// TIA Portal project "Project34" (V11)

(* hardware
DEVICE "S7-400 station_1"  S7400.Device
   slot 0: "UR1_0"  UR1  6ES7 400-1TA01-0AA0
   slot 2: "PLC_1"  Unspecific CPU S7 400  6ES7 4XX XXXXX XXXX
*)

// ===== PLC "PLC_1"  Unspecific CPU S7 400 =====

VAR_GLOBAL   // PLC tag table "Default tag table"
   "s1" AT %I0.0 : Bool;
   "s2" AT %I0.1 : Bool;
   "k2" AT %Q0.3 : Bool;
   "b2" AT %I0.3 : Bool;
   "k1" AT %Q0.2 : Bool;
   "Tag_1" AT %T1 : Timer;
   "b1" AT %I0.2 : Bool;
   "Tag_3" AT %T2 : Timer;
   "h1" AT %Q0.0 : Bool;
   "h2" AT %Q0.1 : Bool;
END_VAR

ORGANIZATION_BLOCK "Main"   // OB1, LAD
TITLE = "Main Program Sweep (Cycle)"
{ S7_Optimized_Access := 'FALSE' }
VERSION : 0.1
   VAR_TEMP
      OB1_EV_CLASS : Byte;   // Bits 0-3 = 1 (Coming event), Bits 4-7 = 1 (Event class 1)
      OB1_SCAN_1 : Byte;   // 1 (Cold restart scan 1 of OB 1), 3 (Scan 2-n of OB 1)
      OB1_PRIORITY : Byte;   // Priority of OB Execution
      OB1_OB_NUMBR : Byte;   // 1 (Organization block 1, OB1)
      OB1_RESERVED_1 : Byte;   // Reserved for system
      OB1_RESERVED_2 : Byte;   // Reserved for system
      OB1_PREV_CYCLE : Int;   // Cycle time of previous OB1 scan (milliseconds)
      OB1_MIN_CYCLE : Int;   // Minimum cycle time of OB1 (milliseconds)
      OB1_MAX_CYCLE : Int;   // Maximum cycle time of OB1 (milliseconds)
      OB1_DATE_TIME : Date_And_Time;   // Date and time OB1 started
   END_VAR
   VAR_TEMP   // added for the SCL form of the ladder/FBD networks
      _w1 : Bool;
      _s5time1 : S5Time;
   END_VAR
BEGIN

REGION Network 1
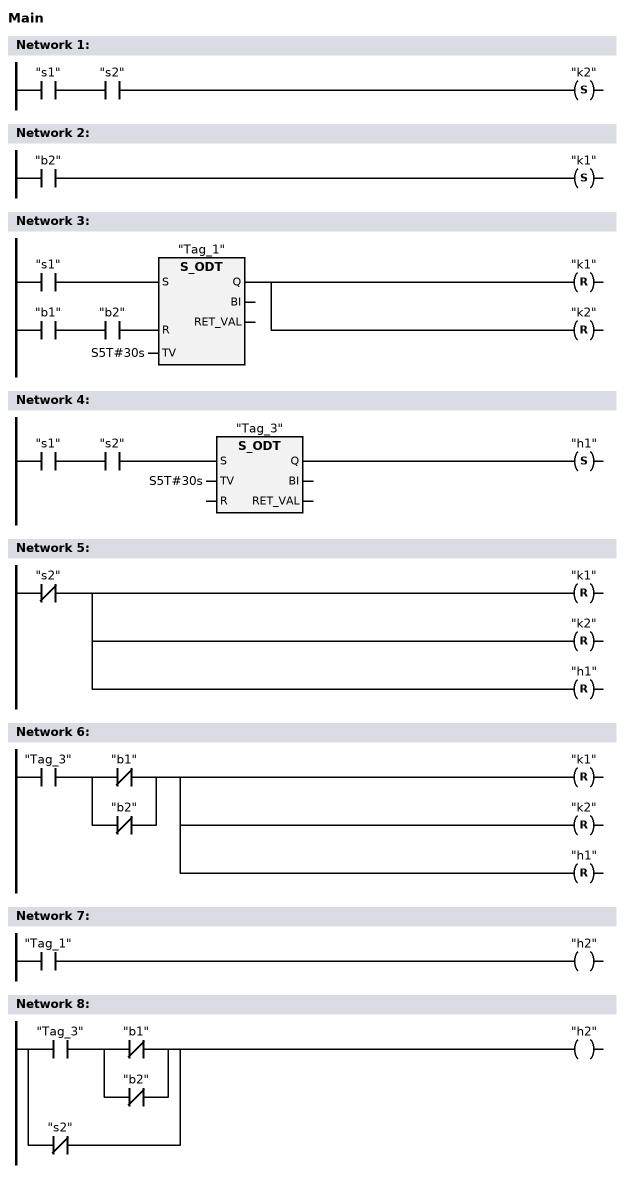
   RUNG wire#powerrail
      Contact( "s1" )
      Contact( "s2" )
      S_Coil( "k2" )
   END_RUNG
   // the same network as SCL:
   IF "s1" AND "s2" THEN "k2" := TRUE; END_IF;
END_REGION

REGION Network 2
   RUNG wire#powerrail
      Contact( "b2" )
      S_Coil( "k1" )
   END_RUNG
   // the same network as SCL:
   IF "b2" THEN "k1" := TRUE; END_IF;
END_REGION

REGION Network 3
   RUNG wire#powerrail
      Contact( "s1" )
      S_ODT(T_NO := "Tag_1", R := wire#w1, TV := S5T#30s, BI =>, RET_VAL =>)
      wire#w2
      R_Coil( "k1" )
   END_RUNG
   RUNG wire#powerrail
      Contact( "b1" )
      Contact( "b2" )
   END_RUNG wire#w1
   RUNG wire#w2
      R_Coil( "k2" )
   END_RUNG
   // the same network as SCL:
   #_s5time1 := S_ODT(T_NO := "Tag_1", S := "s1", R := "b1" AND "b2", TV := S5T#30s, Q => #_w1);
   IF #_w1 THEN
       "k1" := FALSE;
       "k2" := FALSE;
   END_IF;
END_REGION

REGION Network 4
   RUNG wire#powerrail
      Contact( "s1" )
      Contact( "s2" )
      S_ODT(T_NO := "Tag_3", TV := S5T#30s, R :=, BI =>, RET_VAL =>)
      S_Coil( "h1" )
   END_RUNG
   // the same network as SCL:
   #_s5time1 := S_ODT(T_NO := "Tag_3", S := "s1" AND "s2", TV := S5T#30s, Q => #_w1);
   IF #_w1 THEN "h1" := TRUE; END_IF;
END_REGION

REGION Network 5
   RUNG wire#powerrail
      I_Contact( "s2" )
      wire#w1
      R_Coil( "k1" )
   END_RUNG
   RUNG wire#w1
      R_Coil( "k2" )
   END_RUNG
   RUNG wire#w1
      R_Coil( "h1" )
   END_RUNG
   // the same network as SCL:
   IF NOT "s2" THEN
       "k1" := FALSE;
       "k2" := FALSE;
       "h1" := FALSE;
   END_IF;
END_REGION

REGION Network 6
   RUNG wire#powerrail
      Contact( "Tag_3" )
      wire#w1
      I_Contact( "b1" )
      wire#w2
      R_Coil( "k1" )
   END_RUNG
   RUNG wire#w1
      I_Contact( "b2" )
   END_RUNG wire#w2
   RUNG wire#w2
      R_Coil( "k2" )
   END_RUNG
   RUNG wire#w2
      R_Coil( "h1" )
   END_RUNG
   // the same network as SCL:
   IF "Tag_3" AND (NOT "b1" OR NOT "b2") THEN
       "k1" := FALSE;
       "k2" := FALSE;
       "h1" := FALSE;
   END_IF;
END_REGION

REGION Network 7
   RUNG wire#powerrail
      Contact( "Tag_1" )
      Coil( "h2" )
   END_RUNG
   // the same network as SCL:
   "h2" := "Tag_1";
END_REGION

REGION Network 8
   RUNG wire#powerrail
      Contact( "Tag_3" )
      wire#w1
      I_Contact( "b1" )
      wire#w2
      Coil( "h2" )
   END_RUNG
   RUNG wire#w1
      I_Contact( "b2" )
   END_RUNG wire#w2
   RUNG wire#powerrail
      I_Contact( "s2" )
   END_RUNG wire#w2
   // the same network as SCL:
   "h2" := ("Tag_3" AND (NOT "b1" OR NOT "b2")) OR NOT "s2";
END_REGION
END_ORGANIZATION_BLOCK